(*
SPDX-FileCopyrightText: © 2026 Oleksandr Tiutyk <trofimich@gmail.com>
SPDX-License-Identifier: MIT
License: https://opensource.org/license/mit
*)

(*!
<summary>Exposes this library's compiler-initialized namespace.</summary>
<description>
Internal metadata provider; no cyclic body call is needed. The returned namespace is borrowed read-only
storage.
</description>
*)

{attribute 'no_explicit_call' := 'do not call this POU directly'}
PROGRAM INTERNAL CurrentNamespace
VAR
	{attribute 'hide'} 
	_NamespaceExtractor : NamespaceExtractor;
END_VAR

(*!
<summary>Borrows the compiler-initialized library namespace.</summary>
<description>
Do not modify the referenced storage. Reading does not allocate or transfer ownership.
</description>
*)
{attribute 'monitoring' := 'call'}
PROPERTY Name : REFERENCE TO STRING
GET
Name REF= _NamespaceExtractor.CurrentNamespace;
END_GET
END_PROPERTY

END_PROGRAM

(* stored: Version 1.1.0.1
   POU CurrentNamespace: Id {bd9c4cba-5989-4008-99b8-19e7fb541a9f}, SpecialFunc None
   Property Name: Id {761e5a5a-64a6-45eb-ab89-5f6fa252511d}
   Get Get: Id {4eceaf44-dccc-4bda-9902-eb10c976e01d} *)
